FUNCTION F_AmphosAttenuatorEnable : BOOL
VAR_INPUT
	bAmphosOn : BOOL;
END_VAR
VAR_IN_OUT CONSTANT
	stErrors : ST_ErrorStates;
END_VAR
VAR
END_VAR

// Close the attenuator by default
F_AmphosAttenuatorEnable := FALSE;

// Close attenuator if there is a hardware failure
IF stErrors.bHardwareFailure THEN
	RETURN;
END_IF

// Close attenuator if Amphos is not on
IF NOT bAmphosOn THEN
	RETURN;
END_IF

// Close attenuator if there is a leak on the optical table with amphos on, there is a leak in the OPCPA with the carbide on, or there is a leak under the table
IF stErrors.bLeakOpticalTableAmphosOn OR stErrors.bLeakOpcpaCarbideOn OR stErrors.bLeakUnderTable THEN
	RETURN;
END_IF

// Close attenuator if there is an AmphosMRC01 error
IF stErrors.bAmphosMRC01 THEN
	RETURN;
END_IF

F_AmphosAttenuatorEnable := TRUE;

END_FUNCTION

(* stored: Version 1.1.0.1, ProductVersion 3.1.4020.14
   POU F_AmphosAttenuatorEnable: Id {7ab6d45d-4336-488b-ae1d-ec9e617ae7af}, SpecialFunc None *)
